INTERFACE I_Observer

METHOD Update
VAR_INPUT
	nNewValue		:	USINT;
END_VAR
END_METHOD

END_INTERFACE

(* stored: Version 1.1.0.1, ProductVersion 3.1.4024.12
   Itf I_Observer: Id {ad922435-6e6d-45d3-94ba-ef34a18789aa}
   Method Update: Id {975a63c2-7d49-4b17-9936-5f690435e016} *)
